FUNCTION_BLOCK fbStnDegassCtrl
VAR_INPUT

	bEN								: BOOL;
	bEmergencyStop					: BOOL;
	bVacPumpDeact					: BOOL;
	bDegassPumpDeact				: BOOL;
	bCCHighVacuumSignal			: BOOL;
	bDCHighVacuumSignal			: BOOL;
	bDCLowVacuumSignal				: BOOL;

END_VAR

VAR_OUTPUT
	bDegassInProcess				: BOOL;
	bVacPumpOnOff					: BOOL;
	bDegassPumpOnOff				: BOOL;
(*	bCCVacSuctionValveOnOff			: BOOL;*)
	bDCAirReleaseValveOnOff			: BOOL;
	bDCValveOnOff					: BOOL;
END_VAR

VAR

	bStep1							: BOOL;
	bStep2							: BOOL;
	bStep3							: BOOL;

	TON1							: TON;
	TON2							: TON;
	TON3							: TON;

END_VAR
VAR // added by the converter: edge detectors and wires of the graphical bodies
    _w1 : BOOL;
END_VAR

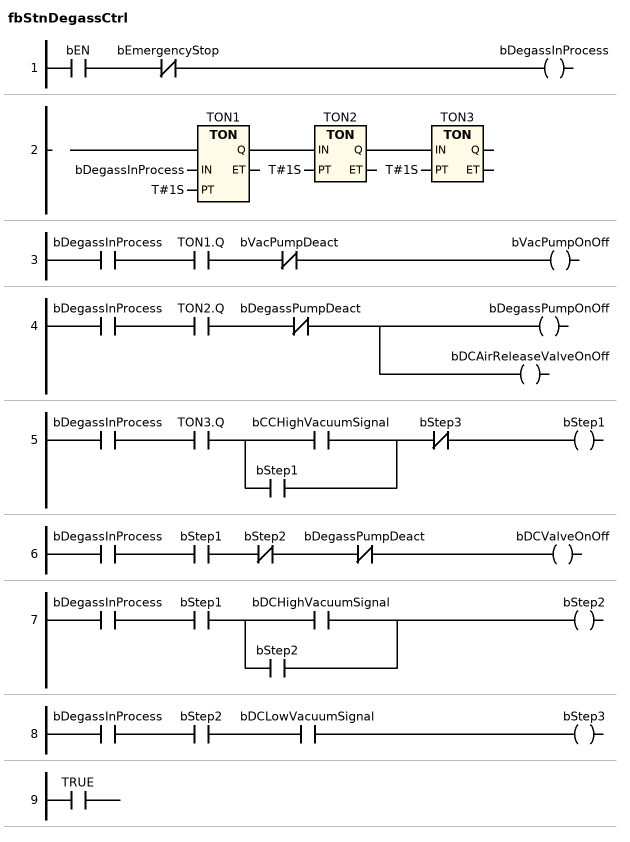
// NETWORK 1
bDegassInProcess := bEN AND NOT bEmergencyStop;

// NETWORK 2
TON1(IN := bDegassInProcess, PT := T#1S); // TON
TON2(IN := TON1.Q, PT := T#1S); // TON
TON3(IN := TON2.Q, PT := T#1S); // TON

// NETWORK 3
bVacPumpOnOff := bDegassInProcess AND TON1.Q AND NOT bVacPumpDeact;

// NETWORK 4
_w1 := bDegassInProcess AND TON2.Q AND NOT bDegassPumpDeact;
bDegassPumpOnOff := _w1;
bDCAirReleaseValveOnOff := _w1;

// NETWORK 5
bStep1 := (bDegassInProcess AND TON3.Q AND (bCCHighVacuumSignal OR bStep1)) AND NOT bStep3;

// NETWORK 6
bDCValveOnOff := bDegassInProcess AND bStep1 AND NOT bStep2 AND NOT bDegassPumpDeact;

// NETWORK 7
bStep2 := bDegassInProcess AND bStep1 AND (bDCHighVacuumSignal OR bStep2);

// NETWORK 8
bStep3 := bDegassInProcess AND bStep2 AND bDCLowVacuumSignal;

// NETWORK 9

END_FUNCTION_BLOCK

(* stored: Version 1.1.0.1, ProductVersion 3.1.4024.12
   POU fbStnDegassCtrl: Id {245d4306-49ee-4efb-8a1d-4299542d9ec4}, SpecialFunc None *)
